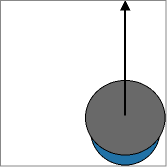
VISUALIZATION VISU_Tube_Top_1  // 167x167
VAR_IN_OUT
	azi : LREAL;
END_VAR
    Ellipse (90,95 70x70)
        p2858320360: azi
    Polygon (85,120) (165,120) (160,135) (90,135)
        p2858320360: azi
    Polygon (120,10) (125,0) (130,10)
        p2858320360: azi
    Ellipse (85,80 80x75)
        p2858320360: azi
    Polyline (125,115) (125,10)
        p2858320360: azi
END_VISUALIZATION

(* stored: Version 1.1.0.1, ProductVersion 3.1.4019.2
   Visu VISU_Tube_Top_1: Id {cc6b7b05-fb4e-4d4a-b7a3-c12b55a9aaa5} *)
